DATA_BLOCK "AutoProcessData_Buffer"
{ S7_Optimized_Access := 'FALSE' }
VERSION : 0.1
// ATTRIBUTES
// AUTO_NUMBER = False
// BLOCK_NUMBER = 1601
// END_ATTRIBUTES
   STRUCT
      DataBuffer { S7_SetPoint := 'False'} : Array[0..55] of "ProcessData";
      DataBuffer_1 { S7_SetPoint := 'False'} : "ProcessData";
      DataBuffer_2 : "ProcessData";
      DataBuffer_3 : "ProcessData";
      DataBuffer_4 : "ProcessData";
      DataBuffer_5 : "ProcessData";
      DataBuffer_6 : "ProcessData";
      VAL { S7_SetPoint := 'True'} : Int;
      SelectButton : Int;
      Button_2 : Bool;
      Button_3 : Bool;
      Button_4 : Bool;
      Button_5 : Bool;
      Button_6 : Bool;
   END_STRUCT;


BEGIN

END_DATA_BLOCK

